// TIA Portal V18 export
FUNCTION_BLOCK "FB_PT_Motors"   // FB2, LAD
{ S7_Optimized_Access := 'TRUE' }
// stored: MemoryReserve 100, SetENOAutomatically false
BEGIN

REGION Network 1: partmotor
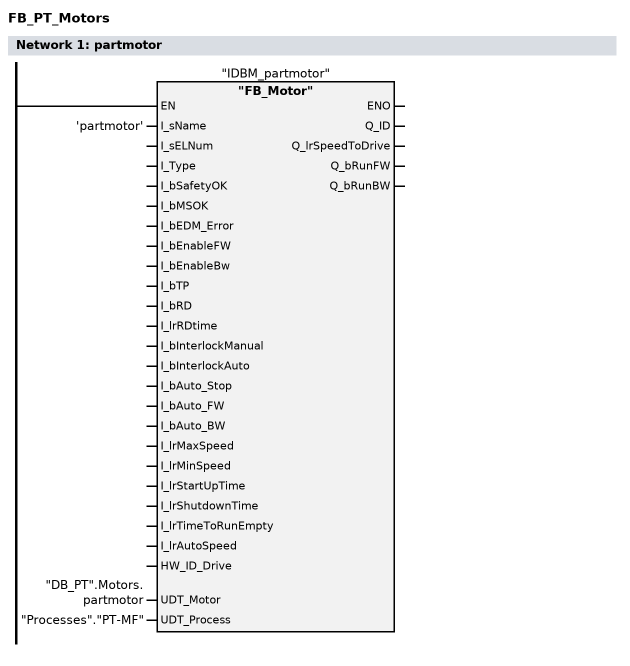
   RUNG wire#powerrail
      "IDBM_partmotor"(I_sName := 'partmotor', I_sELNum :=, I_Type :=, I_bSafetyOK :=, I_bMSOK :=, I_bEDM_Error :=, I_bEnableFW :=, I_bEnableBw :=, I_bTP :=, I_bRD :=, I_lrRDtime :=, I_bInterlockManual :=, I_bInterlockAuto :=, I_bAuto_Stop :=, I_bAuto_FW :=, I_bAuto_BW :=, I_lrMaxSpeed :=, I_lrMinSpeed :=, I_lrStartUpTime :=, I_lrShutdownTime :=, I_lrTimeToRunEmpty :=, I_lrAutoSpeed :=, HW_ID_Drive :=, UDT_Motor := "DB_PT".Motors.partmotor, UDT_Process := "Processes"."PT-MF", Q_ID =>, Q_lrSpeedToDrive =>, Q_bRunFW =>, Q_bRunBW =>)
   END_RUNG
   // the same network as SCL:
   "IDBM_partmotor"(I_sName := 'partmotor',   // "FB_Motor"
                    UDT_Motor := "DB_PT".Motors.partmotor,
                    UDT_Process := "Processes"."PT-MF");
END_REGION
END_FUNCTION_BLOCK
